{attribute 'GeneratedUsingTerminal: EPP1816-3008-0016'}
{attribute addProperty BoxType "EPP1816-3008-0016"}
{attribute addProperty Id "DIG_Inputs_Channel_1AT %I*DIG_Inputs_Channel_38F9DD278DIG_Inputs_Channel_2AT %I*DIG_Inputs_Channel_38F9DD278AI_Inputs_Channel_1AT %I*AI_Inputs_Channel_C3DE7A0A4AI_Inputs_Channel_2AT %I*AI_Inputs_Channel_C3DE7A0A4AI_Inputs_Channel_3AT %I*AI_Inputs_Channel_C3DE7A0A4AI_Inputs_Channel_4AT %I*AI_Inputs_Channel_C3DE7A0A4AI_Inputs_Channel_5AT %I*AI_Inputs_Channel_C3DE7A0A4AI_Inputs_Channel_6AT %I*AI_Inputs_Channel_C3DE7A0A4DIG_Inputs_DeviceAT %I*DIG_Inputs_Device_B3EA42044WcStateAT %I*WcState_9091E0EB2InfoDataAT %I*InfoData_94A18F5E2"}
{attribute addProperty CRC "2452687204"}
{attribute addProperty Size "48"}
TYPE EPP1816_92310964 EXTENDS EtcSlaveTerminalBase_947E5A46 :
STRUCT
	{attribute addProperty Name "DIG_Inputs_Channel_1"}
	DIG_Inputs_Channel_1 : DIG_Inputs_Channel_38F9DD27;
	{attribute addProperty Name "DIG_Inputs_Channel_2"}
	DIG_Inputs_Channel_2 : DIG_Inputs_Channel_38F9DD27;
	{attribute addProperty Name "AI_Inputs_Channel_1"}
	AI_Inputs_Channel_1 : AI_Inputs_Channel_C3DE7A0A;
	{attribute addProperty Name "AI_Inputs_Channel_2"}
	AI_Inputs_Channel_2 : AI_Inputs_Channel_C3DE7A0A;
	{attribute addProperty Name "AI_Inputs_Channel_3"}
	AI_Inputs_Channel_3 : AI_Inputs_Channel_C3DE7A0A;
	{attribute addProperty Name "AI_Inputs_Channel_4"}
	AI_Inputs_Channel_4 : AI_Inputs_Channel_C3DE7A0A;
	{attribute addProperty Name "AI_Inputs_Channel_5"}
	AI_Inputs_Channel_5 : AI_Inputs_Channel_C3DE7A0A;
	{attribute addProperty Name "AI_Inputs_Channel_6"}
	AI_Inputs_Channel_6 : AI_Inputs_Channel_C3DE7A0A;
	{attribute addProperty Name "DIG_Inputs_Device"}
	DIG_Inputs_Device : DIG_Inputs_Device_B3EA4204;
	{attribute addProperty Name "WcState"}
	WcState : WcState_9091E0EB;
	{attribute addProperty Name "InfoData"}
	InfoData : InfoData_94A18F5E;
END_STRUCT
END_TYPE

(* stored: Version 1.2.0.0, ProductVersion 3.1.4024.9
   DUT EPP1816_92310964: Id {84979452-2cec-48a1-abe7-dca1367f5ae0} *)
